// TIA Portal V17 export
// export: Created 2026-04-13T11:12:44.3597411Z, ExportSetting WithDefaults, DisplayName Totally Integrated Automation Portal, DisplayVersion V17 Update 4, DisplayName TIA Portal Openness, DisplayVersion V17 Update 4, DisplayName TIA Portal Version Control Interface, DisplayVersion V17, DisplayName SINAMICS Startdrive Advanced, DisplayVersion V17, DisplayName SINAMICS Startdrive G130, G150, S120, S150, SINAMICS MV, S210, DisplayVersion V17, DisplayName SINAMICS Startdrive G110M, G120, G120C, G120D, G120P, G115D, DisplayVersion V17, DisplayName STEP 7 Professional, DisplayVersion V17 Update 4, DisplayName STEP 7 Safety, DisplayVersion V17, DisplayName WinCC Professional, DisplayVersion V17 Update 4
DATA_BLOCK "A6-模拟量输入_DB"   // DB8
VERSION : 0.1
// stored: AutoNumber true, DBAccessibleFromOPCUA true, DBAccessibleFromWebserver true, InstanceOfName A6-模拟量输入, InstanceOfType FB
"A6-模拟量输入"
   // VAR
   //    进风流量计1 { S7_SetPoint := 'True'} : "0-模拟量输入";
   //    进料流量1 { S7_SetPoint := 'True'} : "0-模拟量输入";
   //    进风压差变送器1 { S7_SetPoint := 'True'} : "0-模拟量输入压差";
   //    出风压差变送器1 { S7_SetPoint := 'True'} : "0-模拟量输入压差";
   //    布袋压差变送器1 { S7_SetPoint := 'True'} : "0-模拟量输入压差";
   //    输送高效压差变送器1 { S7_SetPoint := 'True'} : "0-模拟量输入压差";
   //    进料压力1 { S7_SetPoint := 'True'} : "0-模拟量输入";
   //    塔内压力1 { S7_SetPoint := 'True'} : "0-模拟量输入";
   //    管道压力变送器1 { S7_SetPoint := 'True'} : "0-模拟量输入";
   //    进氮压力1 { S7_SetPoint := 'True'} : "0-模拟量输入";
   //    放空比例反馈1 { S7_SetPoint := 'True'} : "0-模拟量输入";
   //    进风加热比例反馈1 { S7_SetPoint := 'True'} : "0-模拟量输入";
   //    回风加热比例反馈1 { S7_SetPoint := 'True'} : "0-模拟量输入";
   //    雾化油压1 { S7_SetPoint := 'True'} : "0-模拟量输入";
   //    氧含仪11 { S7_SetPoint := 'True'} : "0-模拟量输入";
   //    氧含仪12 { S7_SetPoint := 'True'} : "0-模拟量输入";
   //    一级溶剂液位计1 { S7_SetPoint := 'True'} : "0-模拟量输入";
   //    二级溶剂液位计1 { S7_SetPoint := 'True'} : "0-模拟量输入";
   //    除雾溶剂液位计1 { S7_SetPoint := 'True'} : "0-模拟量输入";
   //    前置水罐液位1 { S7_SetPoint := 'True'} : "0-模拟量输入";
   //    阀岛气压1 { S7_SetPoint := 'True'} : "0-模拟量输入";
   //    T1S : TON_TIME;
   //    YC1 { S7_SetPoint := 'True'} : Real;
   //    延迟1 { S7_SetPoint := 'True'} : "步段延迟";
   //    延迟2 { S7_SetPoint := 'True'} : "步段延迟";
   // END_VAR
BEGIN
END_DATA_BLOCK
